// TIA Portal V19 export
TYPE "OOAx_Ctrl"
// stored: Access Published
   STRUCT
      SafeStop : Bool;   // Emergency stop (device in safe state)
      Rst : Bool;   // Reset alarms
      Homing : Bool;   // Homing command
      MovePlus : Bool;   // Move plus direction command
      MoveMinus : Bool;   // Move minus direction command
      MoveAbsolute : Bool;   // Positioning command
      HomeMode : Int;   // 0=Passive, 1=Active
      HomePosition : LReal;   // Home position (mm)
      MoveAbsTarget : LReal;   // Positioning target (mm)
   END_STRUCT;
END_TYPE
